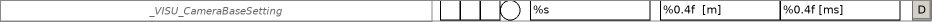
VISUALIZATION _VISU_CameraBase  // 932x22
VAR_IN_OUT
	m_Inst : FB_CameraBase;
END_VAR
    Rectangle (660,0 120x20), "%0.4f [m]", tooltip "TriggerDistance", text variable: m_Inst._fTriggerDistance
        OnMouseDown: write the text variable via Default
    Rectangle (780,0 120x20), "%0.4f [ms]", tooltip "TriggerPulseLength", text variable: m_Inst._fTriggerPulseLength
        OnMouseDown: write the text variable via Default
    RoundedRectangle (440,0 20x20), tooltip "Initialized", colour toggle: m_Inst._bInitialized
    RoundedRectangle (460,0 20x20), tooltip "Camera sink", colour toggle: m_Inst._iCameraSink <> 0
    RoundedRectangle (480,0 20x20), tooltip "Camera trigger", colour toggle: m_Inst._iCameraTrigger <> 0
    Ellipse (500,0 20x20), tooltip "simulate"
        toggle m_Inst._bSimulate
    Frame (0,0 432x22)
        shows _VISU_CameraBaseSetting(m_Inst := m_Inst)
    Button (912,0 20x20), "D", tooltip "Camera Detail: %s", invisible if: m_Inst._sVisuName='unvailable'
        p4168582468: m_Inst._sVisuName
        OnMouseClick: change screen: AssignExpression m_Inst._sVisuName
    Rectangle (530,0 120x20), "%s", tooltip "configured camera mode, active=%s", text variable: m_Inst._eCameraMode
        p4168582468: m_Inst.eCameraMode
        OnMouseDown: write the text variable via Default
END_VISUALIZATION

(* stored: Version 1.1.0.1, ProductVersion 3.1.4024.3
   Visu _VISU_CameraBase: Id {16bd02fb-b1b4-4018-861c-b433b453e903} *)
